Staubli VAL3: Expansion.dtx

mdesc mNomSpeed
num nState
string sFileDelete = "Disk://data/deletedfile"
string sFrom = "Disk://data/copy/1.txt"
string sTo = "Disk://data/copy/copy.txt"
string sFromRename = "Disk://data/rename/1.txt"
string sToRename = "Disk://data/rename/re.txt"
string sFileExist = "Disk://data/exist/exist.txt"
string sFileRead = "Disk://data/fileoperation/read.txt"
num nFileHandler
num nLine
string sLine
string sFileWrite = "Disk://data/fileoperation/write.txt"
num nPwrCnt
num nCircleErr
pointRx pPointIn[4]
  [0] = {fatherId=world[0]}
  [1] = {fatherId=world[0]}
  [2] = {fatherId=world[0]}
  [3] = {fatherId=world[0]}
num nRadius
frame fCircleFrame = {fatherId=world[0]}
jointRx jArmLimit[2]
  [0] = {j1=-100, j2=-50, j3=-50, j4=-100, j5=-60, j6=-100}
  [1] = {j1=150, j2=100, j3=100, j4=100, j5=100, j6=100}
jointRx jCellLimit[2]
  [0] = {j1=-100, j2=-100, j3=-100, j4=-100, j5=-85, j6=-100}
  [1] = {j1=120, j2=120, j3=120, j4=120, j5=90, j6=300}
